{attribute 'qualified_only'}
{attribute 'strict'}
TYPE E_SeqSpeedDoor :
(
	UNKNOWN := 0,
	IDLE,
	OPENING,
	OPENED,
	CLOSING,
	CLOSED,
	ERROR
);
END_TYPE

(* stored: Version 1.1.0.1, ProductVersion 3.1.4024.12
   DUT E_SeqSpeedDoor: Id {cbc7d332-1a91-4874-92fd-8fa482e939f5} *)
